// TwinCAT 3 PLC project Untitled1
// ProgramVersion: 3.1.4024.0
// libraries:
//   Tc2_Standard, * (Beckhoff Automation GmbH)
//   Tc2_System, * (Beckhoff Automation GmbH)
//   Tc3_Mc3PlanarMotion, * (Beckhoff Automation GmbH)
//   Tc3_Module, * (Beckhoff Automation GmbH)
//   Tc3_Physics, * (Beckhoff Automation GmbH)
// project tree:
//   / GlobalTextList.TcGTLO, PlcTask.TcTTO, Visualization Manager.TcVMO (not stored)
//   POUs/ MAIN.TcPOU
//   VISUs/ Visualization.TcVIS, Visu_Variable.TcPOU
// real-time tasks:
//   TASK PlcTask: cycle T#10ms, priority 20, ADS port 350

CONFIGURATION Untitled1
    RESOURCE PLC ON TwinCAT3
        TASK PlcTask(INTERVAL := T#10ms, PRIORITY := 20);
        PROGRAM MAIN WITH PlcTask : MAIN;
        PROGRAM Visu_Variable WITH PlcTask : Visu_Variable;
    END_RESOURCE
END_CONFIGURATION

// ---- POUs/MAIN.TcPOU
PROGRAM MAIN
VAR
	mcMover						: ARRAY [1..ciMoverMax] OF MC_PlanarMover;
	i							: INT;
END_VAR
VAR
	CONSTANT
	ciMoverMax					: INT := 4;
END_VAR

FOR i:= 1 TO ciMoverMax DO
	mcMover[i].Update();
END_FOR

END_PROGRAM

// ---- VISUs/Visu_Variable.TcPOU
PROGRAM Visu_Variable
VAR
	i							: INT;
	stMoverPos					: ARRAY [1..ciMoverMax] OF MoverVector; // Visualizationの画面位置
	stMoverPos_Origin			: ARRAY [1..ciMoverMax] OF MoverVector; // 実位置の確保
	strMoverText				: ARRAY [1..ciMoverMax] OF STRING; // 可動子上に表示される文字列
	strMoverPosText_Num			: ARRAY [1..ciMoverMax] OF STRING; // 可動子番号
	strMoverPosText_x			: ARRAY [1..ciMoverMax] OF STRING; // 可動子のX座標
	strMoverPosText_y			: ARRAY [1..ciMoverMax] OF STRING; // 可動子のY座標
	strMoverPosText_c			: ARRAY [1..ciMoverMax] OF STRING; // 可動子のC座標
END_VAR
VAR
	CONSTANT
	ciMoverMax					: INT := 4;
	ciMoverPos_OffsetX			: LREAL := -200; //Mover番号分かける (i-1)
	ciMoverPos_OffsetY			: LREAL := -200;
END_VAR

FOR i:=1 TO ciMoverMax DO
	//値の登録
	stMoverPos[i] := MAIN.mcMover[i].MCTOPLC.ACT.ActPos; // 可動子の実位置を代入する
	stMoverPos_Origin[i] := stMoverPos[i]; // 内部使用用に確保する
	stMoverPos[i].x := stMoverPos[i].x + ciMoverPos_OffsetX*(i-1); // 原点位置にオフセットする
	stMoverPos[i].y := (-1)*stMoverPos[i].y + ciMoverPos_OffsetY; // 原点位置にオフセットする。Visualizationの画面はYが反転なので-がけする
	stMoverPos[i].c := (-1)*stMoverPos[i].c; //Visualizationと回転方向が逆なので-かける 
	
	//テキストの登録
	strMoverPosText_Num[i] := AddText_MoverNum(iNumber:= i); // 可動子番号登録
	strMoverPosText_x[i] := AddText_MovePos(lrPosition:= stMoverPos_Origin[i].x); // 可動子X座標を登録
	strMoverPosText_y[i] := AddText_MovePos(lrPosition:= stMoverPos_Origin[i].y); // 可動子Y座標を登録
	
	//表示テキストを選択 いらないものはコメントアウト
	strMoverText[i] := ''; //初期化
	strMoverText[i] := CONCAT(strMoverText[i], strMoverPosText_Num[i]); //可動子番号表示
	strMoverText[i] := CONCAT(strMoverText[i], strMoverPosText_x[i]); //可動子X座標表示
	strMoverText[i] := CONCAT(strMoverText[i], strMoverPosText_y[i]); //可動子Y座標表示
END_FOR

METHOD AddText_MovePos : STRING
VAR_INPUT
	lrPosition		: LREAL;
END_VAR
VAR
	strTmpText		: STRING;
END_VAR
strTmpText := LREAL_TO_STRING(lrPosition); //数字をテキストに変換
strTmpText := DELETE(strTmpText, 255, FIND(strTmpText, '.')+2); //小数点1桁以下を削除
AddText_MovePos := CONCAT(strTmpText, '$n'); //改行の追加
END_METHOD

METHOD AddText_MoverNum : STRING
VAR_INPUT
	iNumber				: INT;
END_VAR
AddText_MoverNum := CONCAT(INT_TO_STRING(iNumber), '$n'); //番号を変換して改行を追加
END_METHOD

END_PROGRAM

// ---- GlobalTextList.TcGTLO
TEXTLIST GlobalTextList
  66 = '%s'
  17 = '0'
  787 = '120'
  796 = '240'
  954 = '360'
  789 = '480'
  944 = '600'
  253 = '720'
END_TEXTLIST

// ---- VISUs/Visualization.TcVIS
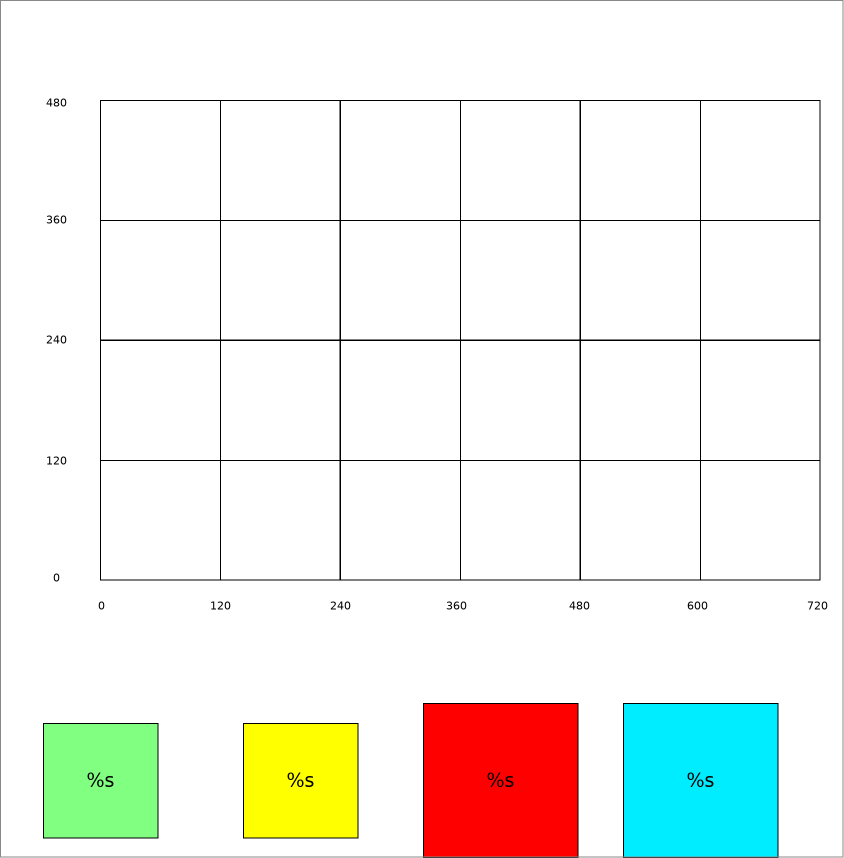
VISUALIZATION Visualization  // 844x858
    Label (75,588 53x36), "0"
    Label (194,588 53x36), "120"
    Label (314,588 53x36), "240"
    Label (430,588 53x36), "360"
    Label (553,588 53x36), "480"
    Label (671,588 53x36), "600"
    Label (791,588 53x36), "720"
    Rectangle (100,100 240x240)
    Rectangle (340,100 240x240)
    Rectangle (580,100 240x240)
    Rectangle (100,340 240x240)
    Rectangle (340,340 240x240)
    Rectangle (580,340 240x240)
    RoundedRectangle (423,703 155x155), "%s", text variable: Visu_Variable.strMoverText[3]
        p3560616238: Visu_Variable.stMoverPos[3].x
        p2738717112: Visu_Variable.stMoverPos[3].y
        p2277200375: Visu_Variable.stMoverPos[3].c
    RoundedRectangle (623,703 155x155), "%s", text variable: Visu_Variable.strMoverText[4]
        p3560616238: Visu_Variable.stMoverPos[4].x
        p2738717112: Visu_Variable.stMoverPos[4].y
        p2277200375: Visu_Variable.stMoverPos[4].c
    RoundedRectangle (43,723 115x115), "%s", text variable: Visu_Variable.strMoverText[1]
        p3560616238: Visu_Variable.stMoverPos[1].x
        p2738717112: Visu_Variable.stMoverPos[1].y
        p2277200375: Visu_Variable.stMoverPos[1].c
    RoundedRectangle (243,723 115x115), "%s", text variable: Visu_Variable.strMoverText[2]
        p3560616238: Visu_Variable.stMoverPos[2].x
        p2738717112: Visu_Variable.stMoverPos[2].y
        p2277200375: Visu_Variable.stMoverPos[2].c
    Line (220,100) (220,580)
    Line (460,100) (460,580)
    Line (700,100) (700,580)
    Line (100,220) (820,220)
    Line (100,460) (820,460)
    Label (30,560 53x36), "0"
    Label (30,443 53x36), "120"
    Label (30,322 53x36), "240"
    Label (30,202 53x36), "360"
    Label (30,85 53x36), "480"
END_VISUALIZATION
